{attribute addProperty BoxType "EP9128-0021-0019"}
{attribute addProperty Id "A_0016_EP9214_0023_0019EP9214_38F98C7664080A_0017_EP9214_0023_0020EP9214_38F98C7664080A_0018_EP9214_0023_0021EP9214_38F98C7664080A_0019_EP9214_0023_0022EP9214_38F98C7664080A_0020_EP9224_0023_0016EP9224_F6E470F9896112A_0021_EP9224_0023_0017EP9224_F6E470F9896112A_0024_EP9521_0020_0000A_0024_EP9521_0020_0000_5317D7A023229A_0022_EP9224_0037_0017A_0022_EP9224_0037_0017_E33DE408162A_0013_EP9128_0021_0019_2_EP9128_1021EP9128_179A0949162A_0013_EP9128_0021_0019_3_EP9128_2021EP9128_179A0949162"}
{attribute addProperty CRC "3914093148"}
{attribute addProperty SizeInBites "4632"}
{attribute addProperty SizeInBytes "579"}
TYPE A_0013_EP9128_0021_0019_E94C525C EXTENDS EP9128_179A0949 :
STRUCT
	{attribute addProperty Name "A_0016_EP9214_0023_0019"}
	A_0016_EP9214_0023_0019 : EP9214_38F98C76;
	{attribute addProperty Name "A_0017_EP9214_0023_0020"}
	A_0017_EP9214_0023_0020 : EP9214_38F98C76;
	{attribute addProperty Name "A_0018_EP9214_0023_0021"}
	A_0018_EP9214_0023_0021 : EP9214_38F98C76;
	{attribute addProperty Name "A_0019_EP9214_0023_0022"}
	A_0019_EP9214_0023_0022 : EP9214_38F98C76;
	{attribute addProperty Name "A_0020_EP9224_0023_0016"}
	A_0020_EP9224_0023_0016 : EP9224_F6E470F9;
	{attribute addProperty Name "A_0021_EP9224_0023_0017"}
	A_0021_EP9224_0023_0017 : EP9224_F6E470F9;
	{attribute addProperty Name "A_0024_EP9521_0020_0000"}
	A_0024_EP9521_0020_0000 : A_0024_EP9521_0020_0000_5317D7A0;
	{attribute addProperty Name "A_0022_EP9224_0037_0017"}
	A_0022_EP9224_0037_0017 : A_0022_EP9224_0037_0017_E33DE408;
	{attribute addProperty Name "A_0013_EP9128_0021_0019_2_EP9128_1021"}
	A_0013_EP9128_0021_0019_2_EP9128_1021 : EP9128_179A0949;
	{attribute addProperty Name "A_0013_EP9128_0021_0019_3_EP9128_2021"}
	A_0013_EP9128_0021_0019_3_EP9128_2021 : EP9128_179A0949;
END_STRUCT
END_TYPE

(* stored: Version 1.2.0.0, ProductVersion 3.1.4024.9
   DUT A_0013_EP9128_0021_0019_E94C525C: Id {3bf61da4-3472-448b-a354-5564e651ec95} *)
